ABB RAPID module: Calibrate_new.mod

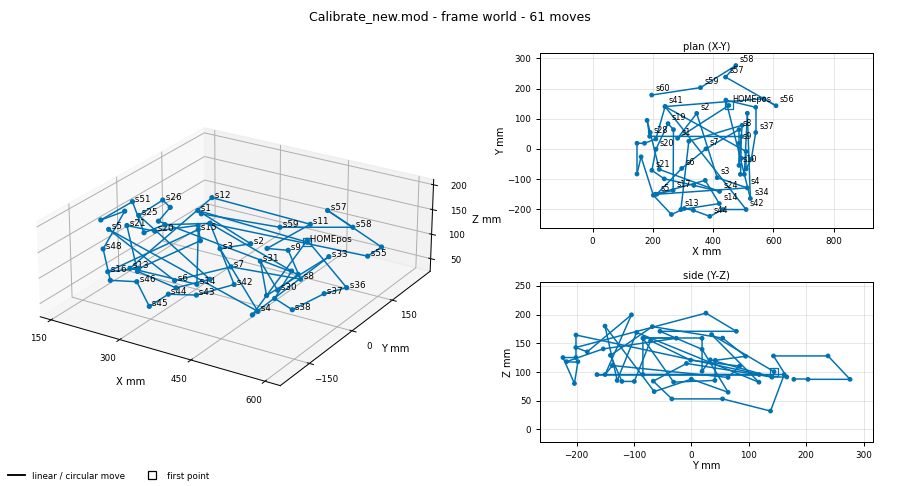
[picture p0: tool path of Calibrate_new.mod in frame world, 61 of 61 moves have a stored position in this frame; points joined in program order, loops and branches not executed]
MODULE Calibrate_new
    CONST robtarget HOMEpos:=[[452.197102023,144.011712884,100.630619004],[0.301166117,0.836912866,-0.428349013,0.159351651],[-1,-3,-2,4],[158.858618137,9E+09,9E+09,9E+09,9E+09,9E+09]];

    CONST robtarget s1:=[[282.1975001,35.092563013,165.269291101],[0.255730755,0.714025669,-0.611615578,0.225156636],[-1,-3,-2,4],[158.858615741,9E+09,9E+09,9E+09,9E+09,9E+09]];
    CONST robtarget s2:=[[345.636867071,117.661303015,82.24910993],[0.096067169,0.752330932,-0.645740984,0.088248796],[-1,-2,-2,4],[158.85861343,9E+09,9E+09,9E+09,9E+09,9E+09]];
    CONST robtarget s3:=[[413.658597024,-95.575640659,168.9569702],[0.099956614,0.780741154,-0.61108647,0.083816774],[-1,-3,-2,4],[155.134281457,9E+09,9E+09,9E+09,9E+09,9E+09]];
    CONST robtarget s4:=[[513.37087898,-129.431296705,85.285254156],[0.099956716,0.780741222,-0.611086464,0.083816065],[-1,-3,-2,4],[155.13428178,9E+09,9E+09,9E+09,9E+09,9E+09]];
    CONST robtarget s5:=[[212.871061955,-150.616545082,180.036028903],[0.085268652,0.672983095,-0.728064139,0.098719905],[-1,-3,-2,4],[155.134279777,9E+09,9E+09,9E+09,9E+09,9E+09]];
    CONST robtarget s6:=[[295.881728898,-64.936748694,65.856721986],[0.085268685,0.672983119,-0.728064193,0.098719317],[-1,-2,-2,4],[175.398367187,9E+09,9E+09,9E+09,9E+09,9E+09]];
    CONST robtarget s7:=[[376.260759153,-0.10158758,87.58293892],[0.085268871,0.672983125,-0.728064242,0.098718756],[-1,-3,-2,4],[175.398372137,9E+09,9E+09,9E+09,9E+09,9E+09]];
    CONST robtarget s8:=[[485.981051386,63.905939855,64.747777214],[0.085268308,0.672982763,-0.728064699,0.098718339],[-1,-3,-2,4],[175.398372458,9E+09,9E+09,9E+09,9E+09,9E+09]];
    CONST robtarget s9:=[[485.981086571,18.620183078,139.555683436],[0.08526845,0.672982687,-0.728064798,0.098718009],[-1,-3,-2,4],[175.398368181,9E+09,9E+09,9E+09,9E+09,9E+09]];
    CONST robtarget s10:=[[485.981652278,-54.804962119,170.951440294],[0.005539815,0.678340248,-0.734622095,0.012417561],[-1,-3,-2,4],[175.398375461,9E+09,9E+09,9E+09,9E+09,9E+09]];
    CONST robtarget s11:=[[496.421669926,78.310559831,170.951187175],[0.005540005,0.678340157,-0.734622184,0.012417189],[-1,-3,-2,4],[175.398368929,9E+09,9E+09,9E+09,9E+09,9E+09]];
    CONST robtarget s12:=[[319.471752161,25.314084465,202.689512175],[0.0055403,0.678340038,-0.734622304,0.012416468],[-1,-3,-2,4],[175.398370839,9E+09,9E+09,9E+09,9E+09,9E+09]];
    CONST robtarget s13:=[[293.171224368,-201.552827985,142.689303651],[0.005540473,0.678339933,-0.734622407,0.012416016],[-2,-3,-2,4],[175.398364908,9E+09,9E+09,9E+09,9E+09,9E+09]];
    CONST robtarget s14:=[[420.532461228,-181.552422587,135.20355933],[0.005540499,0.678339897,-0.734622444,0.012415781],[-2,-3,-2,4],[175.398367814,9E+09,9E+09,9E+09,9E+09,9E+09]];
    CONST robtarget s15:=[[373.977877381,-104.513829124,199.71808832],[0.00554042,0.678339273,-0.734623037,0.012414821],[-1,-3,-2,4],[175.398424972,9E+09,9E+09,9E+09,9E+09,9E+09]];
    CONST robtarget s16:=[[208.270896269,-150.45802031,95.560125593],[0.005540424,0.678339179,-0.734623128,0.012414582],[-1,-2,-2,4],[175.398415749,9E+09,9E+09,9E+09,9E+09,9E+09]];
    CONST robtarget s17:=[[267.500187175,-137.754794121,111.385803855],[0.063312894,-0.696263319,0.712672258,0.057507571],[-1,-2,-2,4],[175.398421455,9E+09,9E+09,9E+09,9E+09,9E+09]];
    CONST robtarget s18:=[[268.527170077,63.864384769,90.521594426],[0.063313028,-0.696263179,0.712672316,0.057508401],[-1,-2,-2,4],[175.398423101,9E+09,9E+09,9E+09,9E+09,9E+09]];
    CONST robtarget s19:=[[250.466640355,83.852399771,110.281460088],[0.089972793,0.693321992,-0.708072227,0.099213067],[-1,-2,-2,4],[175.398425052,9E+09,9E+09,9E+09,9E+09,9E+09]];
    CONST robtarget s20:=[[210.476369487,-1.339579702,120.611028053],[0.048430841,0.69745552,-0.712732048,0.056773923],[-1,-2,-2,4],[175.398426583,9E+09,9E+09,9E+09,9E+09,9E+09]];
    CONST robtarget s21:=[[196.920460095,-71.255644175,154.610868996],[0.048430954,0.697455139,-0.712732441,0.056773574],[-1,-2,-2,4],[175.398420773,9E+09,9E+09,9E+09,9E+09,9E+09]];
    CONST robtarget s22:=[[238.144051758,-99.492153153,83.610664805],[0.036596331,-0.698176273,0.714353085,0.030170677],[-1,-2,-2,4],[175.398425284,9E+09,9E+09,9E+09,9E+09,9E+09]];
    CONST robtarget s23:=[[336.244039752,-121.14409546,83.610275805],[0.036596263,-0.698176245,0.714353095,0.030171181],[-1,-2,-2,4],[175.398423624,9E+09,9E+09,9E+09,9E+09,9E+09]];
    CONST robtarget s24:=[[421.466935022,-141.143734544,129.107288838],[0.036596185,-0.698176245,0.714353085,0.030171511],[-1,-3,-2,4],[175.398422578,9E+09,9E+09,9E+09,9E+09,9E+09]];
    CONST robtarget s25:=[[221.466999029,-68.07971904,179.107194059],[0.03659626,-0.698176248,0.714353075,0.030171583],[-1,-3,-2,4],[175.398423109,9E+09,9E+09,9E+09,9E+09,9E+09]];
    CONST robtarget s26:=[[191.467078601,54.466101628,159.107092984],[0.036596262,-0.69817618,0.714353136,0.030171724],[-1,-3,-2,4],[175.398426217,9E+09,9E+09,9E+09,9E+09,9E+09]];
    CONST robtarget s27:=[[181.002651655,94.467548199,127.436633968],[0.247230319,0.630643887,-0.665467969,0.313556756],[-1,-3,-1,4],[137.746731265,9E+09,9E+09,9E+09,9E+09,9E+09]];
    CONST robtarget s28:=[[189.619455743,41.669843725,120.338666301],[0.144139603,0.661859905,-0.706757227,0.204106498],[-1,-2,-1,4],[137.746735579,9E+09,9E+09,9E+09,9E+09,9E+09]];
    CONST robtarget s29:=[[494.094518272,40.91960118,85.338174445],[0.131028177,0.664579913,-0.710653984,0.190094899],[-1,-3,-1,4],[137.746736064,9E+09,9E+09,9E+09,9E+09,9E+09]];
    CONST robtarget s30:=[[494.094669151,-31.03185753,82.377366547],[0.131028232,0.664579963,-0.710654028,0.190094526],[-1,-3,-1,4],[137.746730055,9E+09,9E+09,9E+09,9E+09,9E+09]];
    CONST robtarget s31:=[[490.473324064,-84.569310669,158.862101089],[0.131028247,0.664580013,-0.71065414,0.190093919],[-1,-2,-1,4],[137.746735805,9E+09,9E+09,9E+09,9E+09,9E+09]];
    CONST robtarget s32:=[[503.623840937,-84.568825175,95.557247475],[0.131028358,0.664579972,-0.71065428,0.190093464],[-1,-3,-1,4],[137.746738987,9E+09,9E+09,9E+09,9E+09,9E+09]];
    CONST robtarget s33:=[[513.624077916,118.104174469,95.556744425],[0.04695928,0.675743803,-0.728837714,0.099803433],[-1,-3,-1,4],[137.746733637,9E+09,9E+09,9E+09,9E+09,9E+09]];
    CONST robtarget s34:=[[523.624116957,-164.629376233,95.55660349],[0.046959298,0.675743732,-0.728837797,0.099803297],[-1,-2,-2,4],[137.746732618,9E+09,9E+09,9E+09,9E+09,9E+09]];
    CONST robtarget s35:=[[442.343497467,161.705071522,95.556426589],[0.046959474,0.67574375,-0.728837811,0.099802996],[-1,-3,-1,4],[137.746732187,9E+09,9E+09,9E+09,9E+09,9E+09]];
    CONST robtarget s36:=[[541.343319041,137.844312633,31.959140511],[0.046959516,0.675743587,-0.72883806,0.099802256],[-1,-3,-1,4],[137.746733471,9E+09,9E+09,9E+09,9E+09,9E+09]];
    CONST robtarget s37:=[[541.343570112,54.268585842,53.152221321],[0.020197521,0.838078155,-0.534284059,0.108432515],[-1,-2,-2,4],[137.74673455,9E+09,9E+09,9E+09,9E+09,9E+09]];
    CONST robtarget s38:=[[526.823024852,-34.145989897,53.151848865],[0.02019662,0.838078042,-0.534284354,0.108432104],[-1,-2,-2,4],[137.746750501,9E+09,9E+09,9E+09,9E+09,9E+09]];
    CONST robtarget s39:=[[509.470342355,-66.453673415,84.040967615],[0.020196654,0.838077943,-0.534284576,0.108431767],[-1,-2,-2,4],[137.746731733,9E+09,9E+09,9E+09,9E+09,9E+09]];
    CONST robtarget s41:=[[240.7544003,140.306701536,91.296812802],[0.034051141,0.740899798,-0.6460004,0.180531141],[-1,-2,-2,4],[-160.61559898,9E+09,9E+09,9E+09,9E+09,9E+09]];
    CONST robtarget s40:=[[509.470330055,-8.628966702,114.918650111],[0.020196725,0.838077933,-0.534284665,0.108431392],[-1,-2,-2,4],[137.746732388,9E+09,9E+09,9E+09,9E+09,9E+09]];
    CONST robtarget s42:=[[509.47030314,-201.234274716,164.47703321],[0.008948963,0.573830481,-0.818096759,0.036826459],[-2,-2,-1,4],[137.746729118,9E+09,9E+09,9E+09,9E+09,9E+09]];
    CONST robtarget s43:=[[432.26981017,-201.233810337,125.204102604],[0.008948703,0.573830332,-0.818096872,0.036826319],[-2,-2,-2,4],[137.746738514,9E+09,9E+09,9E+09,9E+09,9E+09]];
    CONST robtarget s44:=[[389.070712078,-223.904722713,125.203557243],[0.006835909,0.619497518,-0.784083276,0.037276153],[-2,-2,-2,4],[137.746786507,9E+09,9E+09,9E+09,9E+09,9E+09]];
    CONST robtarget s45:=[[334.669695756,-203.90433591,79.991272985],[0.006836098,0.61949739,-0.784083394,0.037275767],[-1,-2,-2,4],[137.746783601,9E+09,9E+09,9E+09,9E+09,9E+09]];
    CONST robtarget s46:=[[304.669750181,-197.836342398,118.044300802],[0.006836224,0.61949725,-0.784083515,0.037275531],[-2,-2,-2,4],[137.746781572,9E+09,9E+09,9E+09,9E+09,9E+09]];
    CONST robtarget s47:=[[261.761637615,-217.836109103,118.044198038],[0.006836329,0.619497206,-0.784083557,0.037275357],[-2,-2,-2,4],[137.74678342,9E+09,9E+09,9E+09,9E+09,9E+09]];
    CONST robtarget s48:=[[201.761783588,-153.775229682,140.286877928],[0.06312954,-0.646976201,0.757761164,0.056872443],[-1,-2,-2,4],[137.746790893,9E+09,9E+09,9E+09,9E+09,9E+09]];
    CONST robtarget s49:=[[161.074561622,-26.366840295,158.846463143],[0.063129328,-0.646975865,0.75776142,0.056873091],[-1,-2,-2,4],[148.548538313,9E+09,9E+09,9E+09,9E+09,9E+09]];
    CONST robtarget s50:=[[147.469444247,-83.464711657,158.846359278],[0.063129773,-0.64697525,0.757761875,0.056873528],[-1,-2,-2,4],[-160.615592721,9E+09,9E+09,9E+09,9E+09,9E+09]];
    CONST robtarget s51:=[[147.469584807,18.542984423,158.846265989],[0.063129718,-0.646975137,0.757761947,0.056873912],[-1,-2,-2,4],[-160.615597846,9E+09,9E+09,9E+09,9E+09,9E+09]];
    CONST robtarget s52:=[[172.331391935,18.543926934,101.297053859],[0.141310514,-0.648254189,0.746824858,0.045282182],[-1,-2,-2,4],[-160.61560025,9E+09,9E+09,9E+09,9E+09,9E+09]];
    CONST robtarget s53:=[[210.070117479,32.748943173,121.296926886],[0.054701,0.661218532,-0.727350568,0.175382455],[-1,-2,-2,4],[-160.615598174,9E+09,9E+09,9E+09,9E+09,9E+09]];
    CONST robtarget s54:=[[240.7544003,140.306701536,91.296812802],[0.034051141,0.740899798,-0.6460004,0.180531141],[-1,-2,-2,4],[-160.61559898,9E+09,9E+09,9E+09,9E+09,9E+09]];
    CONST robtarget s55:=[[568.23779635,166.221485879,91.296516891],[0.034051188,0.740899855,-0.646000509,0.180530507],[-1,-3,-1,4],[-160.61559987,9E+09,9E+09,9E+09,9E+09,9E+09]];
    CONST robtarget s56:=[[608.77236316,143.060318738,128.034476831],[0.03405134,0.740899852,-0.646000626,0.180530069],[-1,-3,-1,4],[-160.615603702,9E+09,9E+09,9E+09,9E+09,9E+09]];
    CONST robtarget s57:=[[441.375800475,238.064372765,128.034127311],[0.034051471,0.740899945,-0.64600072,0.180529331],[-1,-3,-1,4],[-160.615600914,9E+09,9E+09,9E+09,9E+09,9E+09]];
    CONST robtarget s58:=[[475.431971615,276.440290045,87.24480193],[0.022697905,0.779840141,-0.598414046,0.182304113],[-1,-3,-1,4],[-160.615599327,9E+09,9E+09,9E+09,9E+09,9E+09]];
    CONST robtarget s59:=[[358.213688145,203.11989412,87.244498801],[0.022697971,0.779840066,-0.598414379,0.182303333],[-1,-2,-2,4],[-160.615601047,9E+09,9E+09,9E+09,9E+09,9E+09]];
    CONST robtarget s60:=[[196.324801257,178.489029334,87.244487769],[0.011914406,0.813752587,-0.551413872,0.183323526],[0,-2,-2,4],[-178.021474547,9E+09,9E+09,9E+09,9E+09,9E+09]];





    !***********************************************************
    !
    ! Module:  Module1
    !
    ! Description:
    !   <This script is used for sampling>
    !   <Keep the area in front of the Yumi robot empty.>
    !
    ! Author: zlu20001
    !
    ! Version: 1.0
    !
    !***********************************************************


    !***********************************************************
    !
    ! Procedure main
    !
    !   This is the entry point of your program
    !
    !***********************************************************
    PROC calib()
        VAR num rest;
        rest := 5;
        MoveJ HOMEpos,v1000,fine,tool0\WObj:=wobj0;

        WaitTime rest;
        MoveL s1,v1000,fine,tool0\WObj:=wobj0;
        WaitTime rest;
        MoveL s2,v1000,fine,tool0\WObj:=wobj0;
        WaitTime rest;
        MoveL s3,v1000,fine,tool0\WObj:=wobj0;
        WaitTime rest;
        MoveL s4,v1000,fine,tool0\WObj:=wobj0;
        WaitTime rest;
        MoveL s5,v1000,fine,tool0\WObj:=wobj0;
        WaitTime rest;
        MoveL s6,v1000,fine,tool0\WObj:=wobj0;
        WaitTime rest;
        MoveL s7,v1000,fine,tool0\WObj:=wobj0;
        WaitTime rest;
        MoveL s8,v1000,fine,tool0\WObj:=wobj0;
        WaitTime rest;
        MoveL s9,v1000,fine,tool0\WObj:=wobj0;
        WaitTime rest;
        MoveL s10,v1000,fine,tool0\WObj:=wobj0;
        WaitTime rest;
        MoveL s11,v1000,fine,tool0\WObj:=wobj0;
        WaitTime rest;
        MoveL s12,v800,fine,tool0\WObj:=wobj0;
        WaitTime rest;
        MoveL s13,v1000,fine,tool0\WObj:=wobj0;
        WaitTime rest;
        MoveL s14,v1000,fine,tool0\WObj:=wobj0;
        WaitTime rest;
        MoveL s15,v1000,fine,tool0\WObj:=wobj0;
        WaitTime rest;
        MoveL s16,v1000,fine,tool0\WObj:=wobj0;
        WaitTime rest;
        MoveL s17,v1000,fine,tool0\WObj:=wobj0;
        WaitTime rest;
        MoveL s18,v1000,fine,tool0\WObj:=wobj0;
        WaitTime rest;
        MoveL s19,v1000,fine,tool0\WObj:=wobj0;
        WaitTime rest;
        MoveL s20,v1000,fine,tool0\WObj:=wobj0;
        WaitTime rest;
        MoveL s21,v1000,fine,tool0\WObj:=wobj0;
        WaitTime rest;
        MoveL s22,v1000,fine,tool0\WObj:=wobj0;
        WaitTime rest;
        MoveL s23,v1000,fine,tool0\WObj:=wobj0;
        WaitTime rest;
        MoveL s24,v1000,fine,tool0\WObj:=wobj0;
        WaitTime rest;
        MoveL s25,v1000,fine,tool0\WObj:=wobj0;
        WaitTime rest;
        MoveL s26,v1000,fine,tool0\WObj:=wobj0;
        WaitTime rest;
        MoveL s27,v1000,fine,tool0\WObj:=wobj0;
        WaitTime rest;
        MoveL s28,v1000,fine,tool0\WObj:=wobj0;
        WaitTime rest;
        MoveL s29,v1000,fine,tool0\WObj:=wobj0;
        WaitTime rest;
        MoveL s30,v1000,fine,tool0\WObj:=wobj0;
        WaitTime rest;
        MoveL s31,v500,fine,tool0\WObj:=wobj0;
        WaitTime rest;
        MoveL s32,v1000,fine,tool0\WObj:=wobj0;
        WaitTime rest;
        MoveL s33,v1000,fine,tool0\WObj:=wobj0;
        WaitTime rest;
        MoveL s34,v1000,fine,tool0\WObj:=wobj0;
        WaitTime rest;
        MoveL s35,v1000,fine,tool0\WObj:=wobj0;
        WaitTime rest;
        MoveL s36,v1000,fine,tool0\WObj:=wobj0;
        WaitTime rest;
        MoveL s37,v1000,fine,tool0\WObj:=wobj0;
        WaitTime rest;
        MoveL s38,v1000,fine,tool0\WObj:=wobj0;
        WaitTime rest;
        MoveL s39,v1000,fine,tool0\WObj:=wobj0;
        WaitTime rest;
        MoveL s40,v1000,fine,tool0\WObj:=wobj0;
        WaitTime rest;
        MoveL s41,v1000,fine,tool0\WObj:=wobj0;
        WaitTime rest;
        MoveL s42,v1000,fine,tool0\WObj:=wobj0;
        WaitTime rest;
        MoveL s43,v1000,fine,tool0\WObj:=wobj0;
        WaitTime rest;
        MoveL s44,v1000,fine,tool0\WObj:=wobj0;
        WaitTime rest;
        MoveL s45,v1000,fine,tool0\WObj:=wobj0;
        WaitTime rest;
        MoveL s46,v1000,fine,tool0\WObj:=wobj0;
        WaitTime rest;
        MoveL s47,v1000,fine,tool0\WObj:=wobj0;
        WaitTime rest;
        MoveL s48,v1000,fine,tool0\WObj:=wobj0;
        WaitTime rest;
        MoveL s49,v1000,fine,tool0\WObj:=wobj0;
        WaitTime rest;
        MoveL s50,v1000,fine,tool0\WObj:=wobj0;
        WaitTime rest;
        MoveL s51,v1000,fine,tool0\WObj:=wobj0;
        WaitTime rest;
        MoveL s52,v1000,fine,tool0\WObj:=wobj0;
        WaitTime rest;
        MoveL s53,v1000,fine,tool0\WObj:=wobj0;
        WaitTime rest;
        MoveL s54,v1000,fine,tool0\WObj:=wobj0;
        WaitTime rest;
        MoveL s55,v1000,fine,tool0\WObj:=wobj0;
        WaitTime rest;
        MoveL s56,v1000,fine,tool0\WObj:=wobj0;
        WaitTime rest;
        MoveL s57,v1000,fine,tool0\WObj:=wobj0;
        WaitTime rest;
        MoveL s58,v1000,fine,tool0\WObj:=wobj0;
        WaitTime rest;
        MoveL s59,v1000,fine,tool0\WObj:=wobj0;
        WaitTime rest;
        MoveL s60,v1000,fine,tool0\WObj:=wobj0;
        WaitTime rest;


    ENDPROC
ENDMODULE
